TYPE ST_GantryXYZ_Status :
    STRUCT
		CurrentSpeed : LREAL;
    END_STRUCT
END_TYPE

(* stored: Version 1.1.0.1, ProductVersion 3.1.4024.15
   DUT ST_GantryXYZ_Status: Id {0b3a1ebe-92df-461e-ac92-78fbbd4822ef} *)
